// TIA Portal V20 export
TYPE "typeSafetyForcedDoorClose"
// stored: Access Published, IsFailsafeCompliant true, Namespace Safety
   STRUCT
      Door1CloseMemo : Bool;
      Door2CloseMemo : Bool;
      Door3CloseMemo : Bool;
      Door4CloseMemo : Bool;
      Door5CloseMemo : Bool;
      Door6CloseMemo : Bool;
      Door7CloseMemo : Bool;
   END_STRUCT;
END_TYPE
